Staubli VAL3: onRun.pgx

public program onRun(string& x_sItem[])
  local num l_nValue
  local bool l_bOk
  local num l_nIndex
  local num l_nOperator
  local string l_sName
begin
  //
  // decompose
  //
  call saveInOut:decompose_num(x_sItem,l_sName,l_nOperator,l_nValue)
  //
  if l_sName!=""
    // execute
    switch l_nOperator
      case 0,1
        // =
        call setValue(l_nValue,l_sName)
      break
      case 2
        // +1
        call saveInOut:getValue_num(l_nValue,l_sName)
        l_nValue=l_nValue+1
        call setValue(l_nValue,l_sName)
      break
      case 3
        // -1
        call saveInOut:getValue_num(l_nValue,l_sName)
        l_nValue=l_nValue-1
        call setValue(l_nValue,l_sName)
      break
    endSwitch
  endIf
end
